// TIA Portal V19 export
DATA_BLOCK "PPrgArchive7"   // DB507
// stored: IsOnlyStoredInLoadMemory true, MemoryReserve 0, Namespace G
   VAR RETAIN
      PRG : Array[601..700] of "PPrg_Data";
   END_VAR
BEGIN
END_DATA_BLOCK
